Staubli VAL3: outOfRange.pgx

program outOfRange()
  local num i
  local num l_nPoint
  local num l_nStackPoint
  local string l_sMessage
  local string l_sTraj
begin
  // find which trajectory and which point
  wait(isSettled())
  l_sTraj=cycleStatus:sTraj
  //
  l_nPoint=cycleStatus:nPoint
  // call the onEvent
  call OnEvent:OnCycleEvent(11)
  // out of range
  call language:message(l_sMessage,-5)
  l_sMessage=l_sMessage+" "+l_sTraj+" POINT: "+toString("4",l_nPoint)
  popUpMsg(l_sMessage)
  logMsg("[KERNEL] trajectory:POINT OUT OF RANGE, "+l_sTraj+" POINT: "+toString("4",l_nPoint))
  //
end
